// TIA Portal V19 export
TYPE "C205_VAR_IF_CVE_TYPIC"
   STRUCT
      EXT_AUT { ExternalAccessible := 'False'; ExternalVisible := 'False'; ExternalWritable := 'False'} : Bool;   // Externe (hoofd) beveiliging aangesproken
      EXT_HW { ExternalAccessible := 'False'; ExternalVisible := 'False'; ExternalWritable := 'False'} : Bool;   // Sturings hardware (PLC) in storing
      STO { ExternalAccessible := 'False'; ExternalVisible := 'False'; ExternalWritable := 'False'} : Struct   // Opsomming van alle storingen en meldingen
         A001 : Bool;   // Beveiliging aangesproken
         A002 : Bool;   // Storing batterij
      END_STRUCT;
   END_STRUCT;
END_TYPE
